TYPE U_XTS_STATION_CTRL :
UNION
  stCtrl              : ARRAY[1..MAX_STATION] OF ST_STATION_CTRL;

  byCtrl    AT %Q*    : ARRAY[1..MAX_STATION] OF
                        ARRAY[1..SIZEOF(ST_STATION_CTRL)] OF BYTE;
END_UNION
END_TYPE

(* stored: Version 1.1.0.1
   DUT U_XTS_STATION_CTRL: Id {a9e22b61-a73d-4398-bb13-5f61461d2f2d} *)
